FUNCTION_BLOCK BOOL2STRIP (* SIFB *)
  (* Version 0.1, 2009-05-27, 4DIAC-IDE, ACIN *)
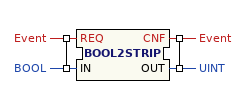
  EVENT_INPUT
    REQ WITH IN; (* Normal Execution Request *)
  END_EVENT
  EVENT_OUTPUT
    CNF WITH OUT; (* Execution Confirmation *)
  END_EVENT
  VAR_INPUT
    IN : BOOL; (* Input event qualifier *)
  END_VAR
  VAR_OUTPUT
    OUT : UINT; (* Output event qualifier *)
  END_VAR
END_FUNCTION_BLOCK
